Staubli VAL3: create.pgx

public program create(string& x_sConveyorList[] (dimensions=1))
  local num l_i
begin
  // Initialize and start conveyor libraries
  //
  // Input Param
  //  x_sConveyorList  : List of conveyors to be created
  //
  // Output param
  //  none       :
  //
  //----------------------------------------------------------------
  //
  call init(x_sConveyorList,nStatus)
  if nStatus==0
    taskCreate sTASK,100,tracking()
  else
    if bAnd(cfg:nLog,cfg:nLOGMISC)==cfg:nLOGMISC
      logMsg(sErrorMessage)
    endIf
    popUpMsg(sErrorMessage)
  endIf
end
